FUNCTION_BLOCK FB_ApplicationMover IMPLEMENTS I_MoverApplication
VAR
	ipMoverStandard	: I_XPlanarMoverStandard;
	
	stProductData	: ST_ProductData;
	
	nMoverIndex		: INT;
	
	nTrackId		: UDINT;
	
	// customer Data
	bIsLoaded		: BOOL;	
		
				
END_VAR

VAR_OUTPUT
	VisuPos	: MoverVector;
END_VAR

METHOD Cycle


VAR_INST
	nTestCounter	: UINT;
END_VAR
IF std <> 0 THEN
	
	nTestCounter := nTestCounter +1;
	
	std.cycle();
	
	VisuPos   := std.P_ActPosition;
	VisuPos.c := std.P_RotationAngleModulo;
			
END_IF
END_METHOD

PROPERTY P_MoverIndex : INT
GET
P_MoverIndex := nMoverIndex;
END_GET
SET
nMoverIndex := P_MoverIndex;
END_SET
END_PROPERTY

PROPERTY P_ProductData : Reference to ST_ProductData
GET
P_ProductData REF= stProductData;
END_GET
SET
stProductData := P_ProductData;
END_SET
END_PROPERTY

PROPERTY P_TrackId : UDINT
GET
P_TrackId := nTrackId;
END_GET
SET
nTrackId := P_TrackId;
END_SET
END_PROPERTY

PROPERTY std : I_XPlanarMoverStandard
GET
IF ipMoverStandard <> 0 THEN
	std := ipMoverStandard;	
END_IF
END_GET
SET
ipMoverStandard := std;
END_SET
END_PROPERTY

END_FUNCTION_BLOCK

(* stored: Version 1.1.0.1, ProductVersion 3.1.4024.9
   POU FB_ApplicationMover: Id {40b5c66d-1fb4-4d55-9f96-3f23301af31f}, SpecialFunc None
   Method Cycle: Id {3db1001d-9da7-43c7-a358-11235832af95}
   Property P_MoverIndex: Id {8b0bebb8-d22b-43e1-ab25-8038159fc710}
   Get Get: Id {6f9fc754-362d-4beb-b50e-e77684f8d50a}
   Set Set: Id {e9f36281-f830-4039-8a28-5be43aca55c3}
   Property P_ProductData: Id {2fbfbc33-cad6-4c1a-b194-3c225a2cf1a2}
   Get Get: Id {4bf4c121-923d-40dd-9c53-7ec22e020235}
   Set Set: Id {d33adc77-a2c9-4f4a-8e6a-c148905050cb}
   Property P_TrackId: Id {bb3a46f6-fd72-439f-b5bc-ae327bc94714}
   Get Get: Id {46b8b84e-3f2c-4789-b5d6-57d0e1a81c42}
   Set Set: Id {d5f18ced-3aa1-4f6f-8451-8cfd636c29e7}
   Property std: Id {74c2e056-88c5-47b5-acb8-9968b5751165}
   Get Get: Id {fdfe9a14-b3ed-40dd-b13f-11a53d96eb71}
   Set Set: Id {75695d29-ba0d-4136-a3f2-f10c3a65b76b} *)
